{attribute 'linkalways'} 
{attribute 'no_explicit_call' := 'This FB is a CLASS and must be accessed using methods or properties'}
{attribute 'enable_dynamic_creation'}
FUNCTION_BLOCK ABSTRACT ArrayDatatypeBase EXTENDS UserDefinedDatatypeBase IMPLEMENTS I_ArrayDatatype
VAR
END_VAR

PROPERTY PUBLIC ABSTRACT BaseDatatype : I_Datatype
GET
END_GET
END_PROPERTY

METHOD PRIVATE CreateEnumError : I_Error
VAR_INPUT
	Enum : T_MAXSTRING;
END_VAR
VAR
	pError : POINTER TO UnknownEnumerationError;
END_VAR
pError := __NEW(UnknownEnumerationError(EnumString := Enum));
CreateEnumError := pError^;
END_METHOD

METHOD PUBLIC ABSTRACT GetElementAsDatatypeByIndex : I_Datatype
VAR_INPUT
	Index : DINT;
END_VAR
END_METHOD

PROPERTY PUBLIC Identifier : T_MAXSTRING
GET
VAR
	baseTypeAsUdt : I_UserDefinedDatatype;
END_VAR
Identifier := Concat('ARRAY [', DINT_TO_STRING(LowerBound));
Identifier := Concat(Identifier,'..');
Identifier := Concat(Identifier, DINT_TO_STRING(UpperBound));
Identifier := Concat(Identifier, '] OF ');

IF BaseDatatype.TryResolveAsUserDefinedDatatype(baseTypeAsUdt) THEN
	Identifier := Concat(Identifier, baseTypeAsUdt.Identifier);
ELSE
	Identifier := Concat(Identifier, BaseDatatype.TypeName);
END_IF
END_GET
END_PROPERTY

PROPERTY PUBLIC Length : UDINT
GET
Length := ABS(UpperBound - LowerBound) + 1;
END_GET
END_PROPERTY

PROPERTY PUBLIC ABSTRACT LowerBound : DINT
GET
END_GET
END_PROPERTY

METHOD PROTECTED ABSTRACT OnSerializeArrayValues
VAR_INPUT
	Serializer : I_Serializer;
END_VAR
END_METHOD

METHOD PROTECTED OnSerializeTypeWith
VAR_INPUT
	Serializer : I_Serializer;
END_VAR
SUPER^.OnSerializeTypeWith(Serializer);
SerializeBaseType(Serializer);
END_METHOD

METHOD PRIVATE SerializeBaseType
VAR_INPUT
	Serializer : I_Serializer;
END_VAR
IF BaseDatatype = 0 THEN
	RETURN;
END_IF

Serializer.AddKey('baseType');
BaseDatatype.SerializeTypeWith(Serializer);
END_METHOD

METHOD PUBLIC SerializeWith
VAR_INPUT
	Serializer : I_Serializer;
END_VAR
Serializer.StartArray();
OnSerializeArrayValues(Serializer);
Serializer.EndArray();
END_METHOD

METHOD PROTECTED ABSTRACT TryDeserializeArrayValues : BOOL
VAR_INPUT
	Deserializer : I_Deserializer;
	Feedback : I_DeserializerFeedback;
END_VAR
END_METHOD

METHOD TryDeserializeFrom : BOOL
VAR_INPUT
	Deserializer : I_Deserializer;
	Feedback : I_DeserializerFeedback;
END_VAR
TryDeserializeFrom := TryDeserializeArrayValues(Deserializer, Feedback);
END_METHOD

METHOD PUBLIC TryResolveAsArrayDatatype : BOOL
VAR_INPUT
	Destination : REFERENCE TO I_ArrayDatatype;
END_VAR
Destination := THIS^;
TryResolveAsArrayDatatype := TRUE;
END_METHOD

PROPERTY PUBLIC TypeName : T_MAXSTRING
GET
TypeName := 'ARRAY';
END_GET
END_PROPERTY

PROPERTY PUBLIC ABSTRACT UpperBound : DINT
GET
END_GET
END_PROPERTY

END_FUNCTION_BLOCK

(* stored: Version 1.1.0.1, ProductVersion 3.1.4024.13
   POU ArrayDatatypeBase: Id {991b8878-a517-02d7-2a23-e8a5c4d992bd}, SpecialFunc None
   Folder Private: Id {a0b3f2c8-538b-0d38-2337-b28ef79dc85d}
   Folder Protected: Id {63cbfb38-749c-0fb5-2a44-a437ca7a7a1f}
   Property BaseDatatype: Id {e7cc5988-3f2b-0d88-33df-f9d96da8e186}
   Get Get: Id {d831321b-2565-0f88-0f30-441c93e1dfda}
   Method CreateEnumError: Id {939e184c-64cf-002a-3378-ba72004e5620}
   Method GetElementAsDatatypeByIndex: Id {72faebb8-2123-0fbb-3cbb-f1f40ed95eb1}
   Property Identifier: Id {2fb82553-7435-463b-94b6-edc871a50638}
   Get Get: Id {3f40e6ca-bcce-4ae5-ab8f-039359f2d5b2}
   Property Length: Id {c8df4437-652c-04b8-35c6-4856f897a24a}
   Get Get: Id {a600413a-c09c-0e5c-1f92-3e6a4da4c8af}
   Property LowerBound: Id {43a0e3e3-ac35-0ef5-2f1e-26f71eb718d0}
   Get Get: Id {56ab5231-520a-0a94-1273-57edd813d82b}
   Method OnSerializeArrayValues: Id {9b19600a-3aab-0e34-2593-3ab26ca49a5c}
   Method OnSerializeTypeWith: Id {1912559b-ea52-07bd-3eb2-f36f75f918bc}
   Method SerializeBaseType: Id {17ec54ac-5ca8-0857-3bd8-63d2ae8f5f0d}
   Method SerializeWith: Id {684d239f-36a7-0f60-36e3-867125d46b0d}
   Method TryDeserializeArrayValues: Id {c71a1318-b78e-07d7-099f-0801c70cb09d}
   Method TryDeserializeFrom: Id {02cc8c70-2927-0c70-1010-8e0f185e7fac}
   Method TryResolveAsArrayDatatype: Id {36f0ff38-3d27-0156-1669-e3996fafb148}
   Property TypeName: Id {51bf05b3-954f-0c7d-072e-7f4beab269b3}
   Get Get: Id {3101e7aa-7e80-06b0-0ff0-1ad591f00d35}
   Property UpperBound: Id {14db03ff-dba9-0e53-21e8-bc01b8e34fca}
   Get Get: Id {9e0fc847-9fa4-01ae-0e26-6e4d01cd70c0} *)
